FUNCTION_BLOCK Reset3
VAR_INPUT
END_VAR
VAR_OUTPUT
	bResetDone : BOOL;
	bResetError: BOOL;
END_VAR
VAR
	fbReset : MC_Reset;
	ResetOut: ST_McOutputs;
	fbMoveRelative: MC_MoveRelative;
	RelativeOut : ST_McOutputs;
	nState : INT;
END_VAR

CASE nState OF
	
0:
	bResetDone := FALSE;
	fbReset(
		Axis:= GVL.ConveyerAxis, 
		Execute:= TRUE, 
		Done=> ResetOut.Done, 
		Busy=> ResetOut.Busy, 
		Error=> ResetOut.Error, 
		ErrorID=> ResetOut.ErrorID);
		IF NOT fbReset.Error THEN
			nState := 1;
		ELSE
			nState := 999;
		END_IF
1:
	fbMoveRelative(
		Axis:= GVL.ConveyerAxis, 
		Execute:= TRUE, 
		Distance:= 16,
		Done=> RelativeOut.Done, 
		Busy=> RelativeOut.Busy, 
		Active=> RelativeOut.Active, 
		CommandAborted=> RelativeOut.CommandAborted, 
		Error=> RelativeOut.Error, 
		ErrorID=> RelativeOut.ErrorID);
		IF NOT fbMoveRelative.Error THEN
			nState := 2;
		ELSE
			nState := 999;
		END_IF
2:
	bResetDone := TRUE;
	nState := 0;
	
999:
	IF NOT fbMoveRelative.Error AND NOT fbReset.Error THEN
		nState := 0;
		bResetError := FALSE;
	ELSE
		bResetError := TRUE;
	END_IF
END_CASE

END_FUNCTION_BLOCK

(* stored: Version 1.1.0.1, ProductVersion 3.1.4024.11
   POU Reset3: Id {597c4e31-3a66-476b-85d2-28696bcee506}, SpecialFunc None *)
